FUNCTION F_INIT_ST_AnyType : HResult
VAR_INPUT
	stAnyType : POINTER TO MPM_JsonParser.ST_AnyType_User;
END_VAR
VAR
	pBytePointer : POINTER TO BYTE;
END_VAR

IF stAnyType = 0 THEN
	F_INIT_ST_AnyType := MPM_FBResult.E_Result.S_FAILED;
	RETURN;
END_IF
IF stAnyType^.pvalue > 0 THEN
	F_INIT_ST_AnyType := MPM_FBResult.E_Result.S_FAILED;
	RETURN;
END_IF
CASE stAnyType^.typeclass OF
	MPM_JsonParser.E_TypeClassEx.TYPE_BOOL:
		stAnyType^.pvalue := __NEW(BOOL);	
		stAnyType^.diSize := SIZEOF(BOOL);
		F_INIT_ST_AnyType := MPM_FBResult.E_Result.S_OK;
	MPM_JsonParser.E_TypeClassEx.TYPE_BYTE:
		stAnyType^.pvalue := __NEW(BYTE);	
		stAnyType^.diSize := SIZEOF(BYTE);	
		F_INIT_ST_AnyType := MPM_FBResult.E_Result.S_OK;
	MPM_JsonParser.E_TypeClassEx.TYPE_LREAL:
		stAnyType^.pvalue := __NEW(LREAL);	
		stAnyType^.diSize := SIZEOF(LREAL);	
		F_INIT_ST_AnyType := MPM_FBResult.E_Result.S_OK;		
	MPM_JsonParser.E_TypeClassEx.TYPE_DINT:
		stAnyType^.pvalue := __NEW(DINT);	
		stAnyType^.diSize := SIZEOF(DINT);	
		F_INIT_ST_AnyType := MPM_FBResult.E_Result.S_OK;
	MPM_JsonParser.E_TypeClassEx.TYPE_LINT:
		stAnyType^.pvalue := __NEW(LINT);	
		stAnyType^.diSize := SIZEOF(LINT);
		F_INIT_ST_AnyType := MPM_FBResult.E_Result.S_OK;	
	MPM_JsonParser.E_TypeClassEx.TYPE_UDINT:
		stAnyType^.pvalue := __NEW(UDINT);	
		stAnyType^.diSize := SIZEOF(UDINT);
		F_INIT_ST_AnyType := MPM_FBResult.E_Result.S_OK;	
	MPM_JsonParser.E_TypeClassEx.TYPE_INT:
		stAnyType^.pvalue := __NEW(INT);	
		stAnyType^.diSize := SIZEOF(INT);
		F_INIT_ST_AnyType := MPM_FBResult.E_Result.S_OK;		
	MPM_JsonParser.E_TypeClassEx.TYPE_REAL:
		stAnyType^.pvalue := __NEW(REAL);	
		stAnyType^.diSize := SIZEOF(REAL);	
		F_INIT_ST_AnyType := MPM_FBResult.E_Result.S_OK;		
	MPM_JsonParser.E_TypeClassEx.TYPE_WORD:
		stAnyType^.pvalue := __NEW(WORD);	
		stAnyType^.diSize := SIZEOF(WORD);	
		F_INIT_ST_AnyType := MPM_FBResult.E_Result.S_OK;		
	ELSE
		F_INIT_ST_AnyType := MPM_FBResult.E_Result.S_FAILED;				
END_CASE

END_FUNCTION

(* stored: Version 1.1.0.1, ProductVersion 3.1.4024.12
   POU F_INIT_ST_AnyType: Id {6439665d-665c-4d60-a625-eb3fa3d91c45}, SpecialFunc None *)
